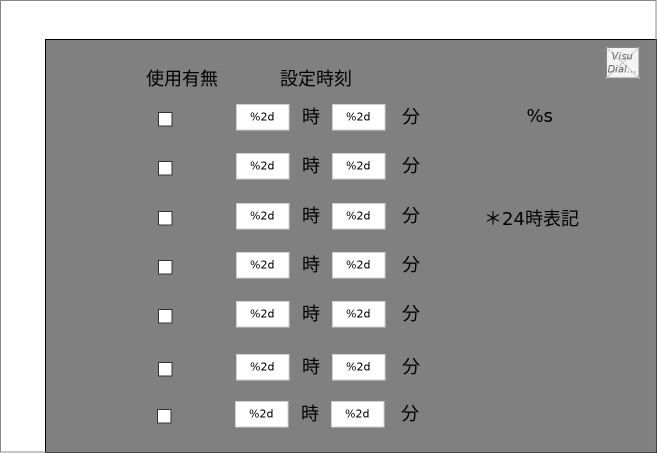
VISUALIZATION d_sampleSchedule  // 657x453
    Rectangle (45,39 612x414)
    Image (606,47 33x31), image: VisuDialogs.ImagePoolDialogs.Delete
        OnMouseClick: CloseDialog Dialog=d_sampleSchedule, Result=OK, NumpadKeypadSet=True
    Textfield (236,104 53x26), "%2d", text variable: gvl_visu.var_scheduleTimeH[0]
        OnMouseClick: write gvl_visu.var_scheduleTimeH[0] via VisuDialogs.Numpad, min 0, max 23
    Textfield (332,104 53x26), "%2d", text variable: gvl_visu.var_scheduleTimeM[0]
        OnMouseClick: write gvl_visu.var_scheduleTimeM[0] via VisuDialogs.Numpad, min 0, max 59
    Checkbox (156,104 27x30), variable: gvl_visu.var_enableSchedule[0]
    Label (291,104 40x26), "時"
    Label (391,104 40x26), "分"
    Label (253,66 126x26), "設定時刻"
    Label (119,66 126x26), "使用有無"
    Textfield (236,153 53x26), "%2d", text variable: gvl_visu.var_scheduleTimeH[1]
        OnMouseClick: write gvl_visu.var_scheduleTimeH[1] via VisuDialogs.Numpad, min 0, max 23
    Textfield (332,153 53x26), "%2d", text variable: gvl_visu.var_scheduleTimeM[1]
        OnMouseClick: write gvl_visu.var_scheduleTimeM[1] via VisuDialogs.Numpad, min 0, max 59
    Checkbox (156,153 27x30), variable: gvl_visu.var_enableSchedule[1]
    Label (291,153 40x26), "時"
    Label (391,153 40x26), "分"
    Textfield (236,203 53x26), "%2d", text variable: gvl_visu.var_scheduleTimeH[2]
        OnMouseClick: write gvl_visu.var_scheduleTimeH[2] via VisuDialogs.Numpad, min 0, max 23
    Textfield (332,203 53x26), "%2d", text variable: gvl_visu.var_scheduleTimeM[2]
        OnMouseClick: write gvl_visu.var_scheduleTimeM[2] via VisuDialogs.Numpad, min 0, max 59
    Checkbox (156,203 27x30), variable: gvl_visu.var_enableSchedule[2]
    Label (291,203 40x26), "時"
    Label (391,203 40x26), "分"
    Textfield (236,252 53x26), "%2d", text variable: gvl_visu.var_scheduleTimeH[3]
        OnMouseClick: write gvl_visu.var_scheduleTimeH[3] via VisuDialogs.Numpad, min 0, max 23
    Textfield (332,252 53x26), "%2d", text variable: gvl_visu.var_scheduleTimeM[3]
        OnMouseClick: write gvl_visu.var_scheduleTimeM[3] via VisuDialogs.Numpad, min 0, max 59
    Checkbox (156,252 27x30), variable: gvl_visu.var_enableSchedule[3]
    Label (291,252 40x26), "時"
    Label (391,252 40x26), "分"
    Textfield (236,301 53x26), "%2d", text variable: gvl_visu.var_scheduleTimeH[4]
        OnMouseClick: write gvl_visu.var_scheduleTimeH[4] via VisuDialogs.Numpad, min 0, max 23
    Textfield (332,301 53x26), "%2d", text variable: gvl_visu.var_scheduleTimeM[4]
        OnMouseClick: write gvl_visu.var_scheduleTimeM[4] via VisuDialogs.Numpad, min 0, max 59
    Checkbox (156,301 27x30), variable: gvl_visu.var_enableSchedule[4]
    Label (291,301 40x26), "時"
    Label (391,301 40x26), "分"
    Textfield (236,354 53x26), "%2d", text variable: gvl_visu.var_scheduleTimeH[5]
        OnMouseClick: write gvl_visu.var_scheduleTimeH[5] via VisuDialogs.Numpad, min 0, max 23
    Textfield (332,354 53x26), "%2d", text variable: gvl_visu.var_scheduleTimeM[5]
        OnMouseClick: write gvl_visu.var_scheduleTimeM[5] via VisuDialogs.Numpad, min 0, max 59
    Checkbox (156,354 27x30), variable: gvl_visu.var_enableSchedule[5]
    Label (291,354 40x26), "時"
    Label (391,354 40x26), "分"
    Textfield (235,401 53x26), "%2d", text variable: gvl_visu.var_scheduleTimeH[6]
        OnMouseClick: write gvl_visu.var_scheduleTimeH[6] via VisuDialogs.Numpad, min 0, max 23
    Textfield (331,401 53x26), "%2d", text variable: gvl_visu.var_scheduleTimeM[6]
        OnMouseClick: write gvl_visu.var_scheduleTimeM[6] via VisuDialogs.Numpad, min 0, max 59
    Checkbox (155,401 27x30), variable: gvl_visu.var_enableSchedule[6]
    Label (290,401 40x26), "時"
    Label (390,401 40x26), "分"
    Label (455,206 153x26), "＊24時表記"
    RoundedRectangle (426,101 228x30), "%s", text variable: gvl_visu.var_DT
END_VISUALIZATION

(* stored: Version 1.1.0.1, ProductVersion 3.1.4024.12
   Visu d_sampleSchedule: Id {9b4482d8-58cc-439a-807c-617e0f564fa3} *)
